FUNCTION F_MatIdtoStr : STRING(20)
VAR_INPUT
	materialId:DINT;
END_VAR
VAR
	i:UINT;
	s1: STRING;
END_VAR

FOR i :=1 TO GVLConst.uiLastMaterialPossible DO
	IF G_DBConn.aMaterialAvailable[i].ID = materialId AND materialId <> 0 THEN
		s1:=G_Dbconn.aMaterialAvailable[i].matId;
		EXIT;
	ELSIF materialId =  0 THEN
		s1:='';
		EXIT;
	END_IF
END_FOR
F_MatIdtoStr:=s1;

END_FUNCTION

(* stored: Version 1.1.0.1, ProductVersion 3.1.4024.12
   POU F_MatIdtoStr: Id {4576843d-0448-477f-9ee4-6a8dac73dcc5}, SpecialFunc None *)
